TYPE (* IEC 61131-3-2.3.3.1 *)
  (* Standard: 61131-3 *)
  (* Version 0.2, 2000-05-16, JHC, Rockwell Automation, File type changed to ".dtp" *)
  (* Version 0.1, 2000-05-10, JHC, Rockwell Automation, Corrected encoding of values. *)
  (* Compiler header: package fb.rt.ita; *)
  (* Compiler Java IBM VisualAge 3.0 *)
  (* ASN.1 tag PRIVATE 12 *)
  ANALOG_SIGNAL_TYPE : (
    SINGLE_ENDED,
    DIFFERENTIAL
  );
END_TYPE
